{attribute 'hide_all_locals'}
FUNCTION_BLOCK PUBLIC FB_FullTimeEmployee IMPLEMENTS I_Employee
VAR_INPUT
END_VAR
VAR_OUTPUT
END_VAR
VAR
	nPersonnelNumberBacking :	UINT;
	sFirstNameBacking		:	STRING;
	sLastNameBacking		:	STRING;	

	nAnnualSalaryBacking	:	UINT;
END_VAR

METHOD GetFullName : STRING
VAR_INPUT
END_VAR
GetFullName := CONCAT(CONCAT(CONCAT(CONCAT(TO_STRING(nPersonnelNumber), ': '), sFirstName), ' '), sLastName);
END_METHOD

METHOD PUBLIC GetMonthlySalary : LREAL
VAR_INPUT
END_VAR
GetMonthlySalary := nAnnualSalary / 12;
END_METHOD

{attribute 'monitoring' := 'variable'}
PROPERTY PUBLIC nAnnualSalary : UINT
GET
nAnnualSalary := nAnnualSalaryBacking;
END_GET
SET
nAnnualSalaryBacking := nAnnualSalary;
END_SET
END_PROPERTY

{attribute 'monitoring' := 'variable'}
PROPERTY nPersonnelNumber : UINT
GET
nPersonnelNumber := nPersonnelNumberBacking;
END_GET
SET
nPersonnelNumberBacking := nPersonnelNumber;
END_SET
END_PROPERTY

{attribute 'monitoring' := 'variable'}
PROPERTY sFirstName : STRING
GET
sFirstName := sFirstNameBacking;
END_GET
SET
sFirstNameBacking := sFirstName;
END_SET
END_PROPERTY

{attribute 'monitoring' := 'variable'}
PROPERTY sLastName : STRING
GET
sLastName := sLastNameBacking;
END_GET
SET
sLastNameBacking := sLastName;
END_SET
END_PROPERTY

END_FUNCTION_BLOCK

(* stored: Version 1.1.0.1, ProductVersion 3.1.4024.4
   POU FB_FullTimeEmployee: Id {a3fcde26-925a-40bc-9c5d-c909b2dc2c4f}, SpecialFunc None
   Method GetFullName: Id {1f4fc63b-1fa3-4484-87f5-a5d21322a9fd}
   Method GetMonthlySalary: Id {19b65e9d-1ce3-41b1-864d-5a175dc14c55}
   Property nAnnualSalary: Id {ecc488aa-1029-4a23-bad9-42ea4e1652f0}
   Get Get: Id {a7dadd95-79a2-4986-84aa-c6df21296c13}
   Set Set: Id {f0f4c3b1-a73f-44e8-8348-fed696c13ad4}
   Property nPersonnelNumber: Id {74ba115b-80a7-4e0a-a70a-3b03d5267acd}
   Get Get: Id {4052ad52-b85c-4f93-8a1f-ace242d16e0a}
   Set Set: Id {6cb9e4f9-177f-419f-ac26-d270c0a57ca0}
   Property sFirstName: Id {79cc0d18-31f6-45b4-a90c-2388ddcf14e2}
   Get Get: Id {2132b76d-6c9c-44ee-8958-7ec7d57ddf5d}
   Set Set: Id {1d40b48b-9bc7-4ec8-9a3a-6c54b03a601a}
   Property sLastName: Id {64bfffa5-c866-4bd1-a01d-e3022db80328}
   Get Get: Id {29f446ab-b8a7-448a-8d66-439ccbf4c4de}
   Set Set: Id {f23147df-1a67-4f9b-8cae-4ed27b0d61da} *)
